// TIA Portal V15.1 export
// export: Created 2024-05-17T05:38:53.3669201Z, ExportSetting WithDefaults, DisplayName Totally Integrated Automation Portal, DisplayVersion V15.1 Update 5, DisplayName TIA Portal Openness, DisplayVersion V15.1 Update 5, DisplayName SINAMICS Startdrive Advanced, DisplayVersion V15.1, DisplayName G130, G150, S120, S150, SINAMICS MV, S210, DisplayVersion V15.1, DisplayName G110M, G120, G120C, G120D, G120P, DisplayVersion V15.1, DisplayName STEP 7 Professional, DisplayVersion V15.1 Update 5, DisplayName STEP 7 Safety, DisplayVersion V15.1, DisplayName WinCC Professional, DisplayVersion V15.1 Update 5, DisplayName SIMATIC Visualization Architect, DisplayVersion V15.1
FUNCTION_BLOCK "LGBCRComm"   // FB6692, FBD
TITLE = LGBCRComm
{ S7_Optimized_Access := 'TRUE' }
VERSION : 0.1
// stored: AutoNumber false, IsIECCheckEnabled false, IsRetainMemResEnabled false, MemoryReserve 100, SetENOAutomatically False, UDAEnableTagReadback false
   VAR_INPUT
      I_PlcActiveShift { ExternalAccessible := 'False'; ExternalVisible := 'False'; ExternalWritable := 'False'} : Int;
      I_PlcActiveBreak { ExternalAccessible := 'False'; ExternalVisible := 'False'; ExternalWritable := 'False'} : Int;
      I_StnAux01Feedback_Int { ExternalAccessible := 'False'; ExternalVisible := 'False'; ExternalWritable := 'False'} : Int;
      I_StnAux02Feedback_Int { ExternalAccessible := 'False'; ExternalVisible := 'False'; ExternalWritable := 'False'} : Int;
      I_StnAux03Feedback_Int { ExternalAccessible := 'False'; ExternalVisible := 'False'; ExternalWritable := 'False'} : Int;
      I_StnAux04Feedback_Int { ExternalAccessible := 'False'; ExternalVisible := 'False'; ExternalWritable := 'False'} : Int;
      I_StnAux05Feedback_Int { ExternalAccessible := 'False'; ExternalVisible := 'False'; ExternalWritable := 'False'} : Int;
      I_StnAux06Feedback_Int { ExternalAccessible := 'False'; ExternalVisible := 'False'; ExternalWritable := 'False'} : Int;
      I_StnAux07Feedback_DInt { ExternalAccessible := 'False'; ExternalVisible := 'False'; ExternalWritable := 'False'} : DInt;
      I_StnAux08Feedback_DInt { ExternalAccessible := 'False'; ExternalVisible := 'False'; ExternalWritable := 'False'} : DInt;
      I_StnAux09Feedback_DInt { ExternalAccessible := 'False'; ExternalVisible := 'False'; ExternalWritable := 'False'} : DInt;
      I_StnAux10Feedback_DInt { ExternalAccessible := 'False'; ExternalVisible := 'False'; ExternalWritable := 'False'} : DInt;
      I_StnAux11Feedback_DInt { ExternalAccessible := 'False'; ExternalVisible := 'False'; ExternalWritable := 'False'} : DInt;
      I_StnAux12Feedback_DInt { ExternalAccessible := 'False'; ExternalVisible := 'False'; ExternalWritable := 'False'} : DInt;
      I_StnAux13Feedback_Real { ExternalAccessible := 'False'; ExternalVisible := 'False'; ExternalWritable := 'False'} : Real;
      I_StnAux14Feedback_Real { ExternalAccessible := 'False'; ExternalVisible := 'False'; ExternalWritable := 'False'} : Real;
      I_StnAux15Feedback_Real { ExternalAccessible := 'False'; ExternalVisible := 'False'; ExternalWritable := 'False'} : Real;
      I_StnAux16Feedback_Real { ExternalAccessible := 'False'; ExternalVisible := 'False'; ExternalWritable := 'False'} : Real;
      I_StnAux17Feedback_Real { ExternalAccessible := 'False'; ExternalVisible := 'False'; ExternalWritable := 'False'} : Real;
      I_StnAux18Feedback_Real { ExternalAccessible := 'False'; ExternalVisible := 'False'; ExternalWritable := 'False'} : Real;
      C_DelayTimeAlarmC { ExternalAccessible := 'False'; ExternalVisible := 'False'; ExternalWritable := 'False'} : Time;
      C_DelayTimeAlarmD { ExternalAccessible := 'False'; ExternalVisible := 'False'; ExternalWritable := 'False'} : Time;
   END_VAR
   VAR_OUTPUT
      O_StnAux01_Int { ExternalAccessible := 'False'; ExternalVisible := 'False'; ExternalWritable := 'False'} : Int;
      O_StnAux02_Int { ExternalAccessible := 'False'; ExternalVisible := 'False'; ExternalWritable := 'False'} : Int;
      O_StnAux03_Int { ExternalAccessible := 'False'; ExternalVisible := 'False'; ExternalWritable := 'False'} : Int;
      O_StnAux04_Int { ExternalAccessible := 'False'; ExternalVisible := 'False'; ExternalWritable := 'False'} : Int;
      O_StnAux05_Int { ExternalAccessible := 'False'; ExternalVisible := 'False'; ExternalWritable := 'False'} : Int;
      O_StnAux06_Int { ExternalAccessible := 'False'; ExternalVisible := 'False'; ExternalWritable := 'False'} : Int;
      O_StnAux07_DInt { ExternalAccessible := 'False'; ExternalVisible := 'False'; ExternalWritable := 'False'} : DInt;
      O_StnAux08_DInt { ExternalAccessible := 'False'; ExternalVisible := 'False'; ExternalWritable := 'False'} : DInt;
      O_StnAux09_DInt { ExternalAccessible := 'False'; ExternalVisible := 'False'; ExternalWritable := 'False'} : DInt;
      O_StnAux10_DInt { ExternalAccessible := 'False'; ExternalVisible := 'False'; ExternalWritable := 'False'} : DInt;
      O_StnAux11_DInt { ExternalAccessible := 'False'; ExternalVisible := 'False'; ExternalWritable := 'False'} : DInt;
      O_StnAux12_DInt { ExternalAccessible := 'False'; ExternalVisible := 'False'; ExternalWritable := 'False'} : DInt;
      O_StnAux13_Real { ExternalAccessible := 'False'; ExternalVisible := 'False'; ExternalWritable := 'False'} : Real;
      O_StnAux14_Real { ExternalAccessible := 'False'; ExternalVisible := 'False'; ExternalWritable := 'False'} : Real;
      O_StnAux15_Real { ExternalAccessible := 'False'; ExternalVisible := 'False'; ExternalWritable := 'False'} : Real;
      O_StnAux16_Real { ExternalAccessible := 'False'; ExternalVisible := 'False'; ExternalWritable := 'False'} : Real;
      O_StnAux17_Real { ExternalAccessible := 'False'; ExternalVisible := 'False'; ExternalWritable := 'False'} : Real;
      O_StnAux18_Real { ExternalAccessible := 'False'; ExternalVisible := 'False'; ExternalWritable := 'False'} : Real;
   END_VAR
   VAR_IN_OUT
      IO_Modes : "Modes";   // Modes
      IO_DBZMToSv : "SupervisionZM";   // Send to supervision system
      IO_DBSvToZM : "SupervisionZM";   // Recieve from supervision system
   END_VAR
   VAR
      DelayAlarmC { ExternalAccessible := 'False'; ExternalVisible := 'False'; ExternalWritable := 'False'} : TON_TIME;
      DelayAlarmD { ExternalAccessible := 'False'; ExternalVisible := 'False'; ExternalWritable := 'False'} : TON_TIME;
      DelayUpperLevelZSAlarmC { ExternalAccessible := 'False'; ExternalVisible := 'False'; ExternalWritable := 'False'} : TON_TIME;
      DelayUpperLevelZSAlarmD { ExternalAccessible := 'False'; ExternalVisible := 'False'; ExternalWritable := 'False'} : TON_TIME;
      DelayUpperLevelPLCAlarmC { ExternalAccessible := 'False'; ExternalVisible := 'False'; ExternalWritable := 'False'} : TON_TIME;
      DelayUpperLevelPLCAlarmD { ExternalAccessible := 'False'; ExternalVisible := 'False'; ExternalWritable := 'False'} : TON_TIME;
   END_VAR
   VAR_TEMP
      Tmp_StnAux13Feedback_Real : Real;
      Tmp_StnAux14Feedback_Real : Real;
      Tmp_StnAux15Feedback_Real : Real;
      Tmp_StnAux16Feedback_Real : Real;
      Tmp_StnAux17Feedback_Real : Real;
      Tmp_StnAux18Feedback_Real : Real;
      Tmp_StnAux13_Real : Real;
      Tmp_StnAux14_Real : Real;
      Tmp_StnAux15_Real : Real;
      Tmp_StnAux16_Real : Real;
      Tmp_StnAux17_Real : Real;
      Tmp_StnAux18_Real : Real;
   END_VAR
BEGIN

REGION Network 1: **** 8 - Outputs **** Plc ActiveShift
   // Plc ActiveShift
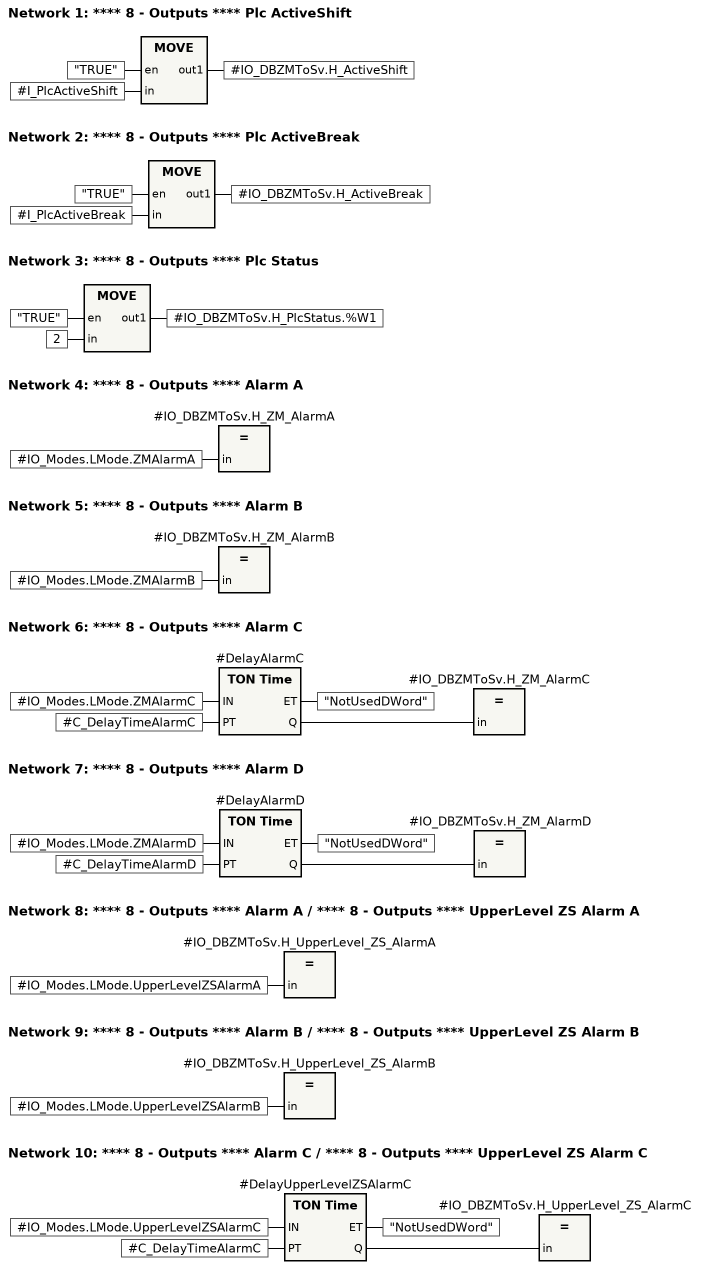
   IF "TRUE" THEN #IO_DBZMToSv.H_ActiveShift := #I_PlcActiveShift; END_IF;
END_REGION

REGION Network 2: **** 8 - Outputs **** Plc ActiveBreak
   // Plc ActiveBreak
   IF "TRUE" THEN #IO_DBZMToSv.H_ActiveBreak := #I_PlcActiveBreak; END_IF;
END_REGION

REGION Network 3: **** 8 - Outputs **** Plc Status
   // Plc Status
   IF "TRUE" THEN #IO_DBZMToSv.H_PlcStatus.%W1 := 2; END_IF;
END_REGION

REGION Network 4: **** 8 - Outputs **** Alarm A
   // Alarm A
   #IO_DBZMToSv.H_ZM_AlarmA := #IO_Modes.LMode.ZMAlarmA;
END_REGION

REGION Network 5: **** 8 - Outputs **** Alarm B
   // Alarm B
   #IO_DBZMToSv.H_ZM_AlarmB := #IO_Modes.LMode.ZMAlarmB;
END_REGION

REGION Network 6: **** 8 - Outputs **** Alarm C
   // Alarm C
   #DelayAlarmC(IN := #IO_Modes.LMode.ZMAlarmC, PT := #C_DelayTimeAlarmC, ET => "NotUsedDWord");   // TON
   #IO_DBZMToSv.H_ZM_AlarmC := #DelayAlarmC.Q;
END_REGION

REGION Network 7: **** 8 - Outputs **** Alarm D
   // Alarm D
   #DelayAlarmD(IN := #IO_Modes.LMode.ZMAlarmD, PT := #C_DelayTimeAlarmD, ET => "NotUsedDWord");   // TON
   #IO_DBZMToSv.H_ZM_AlarmD := #DelayAlarmD.Q;
END_REGION

REGION Network 8: **** 8 - Outputs **** Alarm A / **** 8 - Outputs **** UpperLevel ZS Alarm A
   // Alarm A
   #IO_DBZMToSv.H_UpperLevel_ZS_AlarmA := #IO_Modes.LMode.UpperLevelZSAlarmA;
END_REGION

REGION Network 9: **** 8 - Outputs **** Alarm B / **** 8 - Outputs **** UpperLevel ZS Alarm B
   // Alarm B
   #IO_DBZMToSv.H_UpperLevel_ZS_AlarmB := #IO_Modes.LMode.UpperLevelZSAlarmB;
END_REGION

REGION Network 10: **** 8 - Outputs **** Alarm C / **** 8 - Outputs **** UpperLevel ZS Alarm C
   // Alarm C
   #DelayUpperLevelZSAlarmC(IN := #IO_Modes.LMode.UpperLevelZSAlarmC,   // TON
                           PT := #C_DelayTimeAlarmC,
                           ET => "NotUsedDWord");
   #IO_DBZMToSv.H_UpperLevel_ZS_AlarmC := #DelayUpperLevelZSAlarmC.Q;
END_REGION

REGION Network 11: **** 8 - Outputs **** Alarm D / **** 8 - Outputs **** UpperLevel ZS Alarm D
   // Alarm D
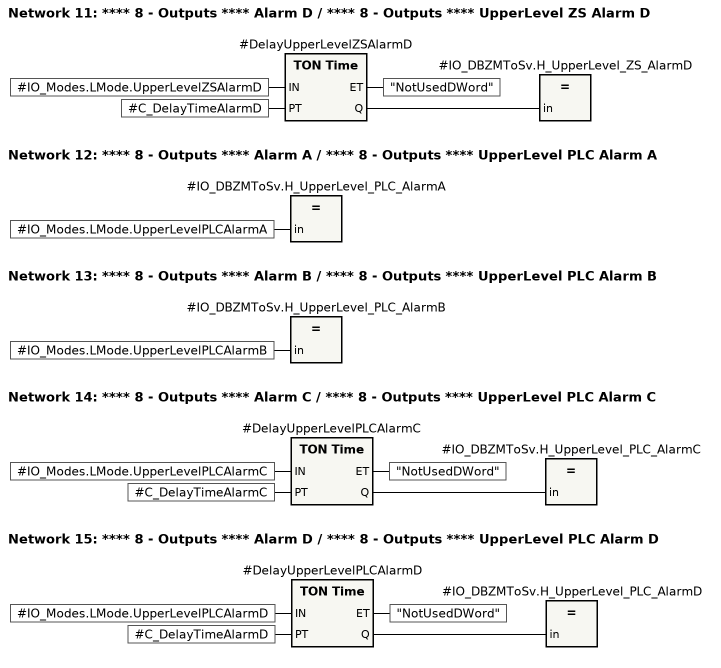
   #DelayUpperLevelZSAlarmD(IN := #IO_Modes.LMode.UpperLevelZSAlarmD,   // TON
                           PT := #C_DelayTimeAlarmD,
                           ET => "NotUsedDWord");
   #IO_DBZMToSv.H_UpperLevel_ZS_AlarmD := #DelayUpperLevelZSAlarmD.Q;
END_REGION

REGION Network 12: **** 8 - Outputs **** Alarm A / **** 8 - Outputs **** UpperLevel PLC Alarm A
   // Alarm A
   #IO_DBZMToSv.H_UpperLevel_PLC_AlarmA := #IO_Modes.LMode.UpperLevelPLCAlarmA;
END_REGION

REGION Network 13: **** 8 - Outputs **** Alarm B / **** 8 - Outputs **** UpperLevel PLC Alarm B
   // Alarm B
   #IO_DBZMToSv.H_UpperLevel_PLC_AlarmB := #IO_Modes.LMode.UpperLevelPLCAlarmB;
END_REGION

REGION Network 14: **** 8 - Outputs **** Alarm C / **** 8 - Outputs **** UpperLevel PLC Alarm C
   // Alarm C
   #DelayUpperLevelPLCAlarmC(IN := #IO_Modes.LMode.UpperLevelPLCAlarmC,   // TON
                           PT := #C_DelayTimeAlarmC,
                           ET => "NotUsedDWord");
   #IO_DBZMToSv.H_UpperLevel_PLC_AlarmC := #DelayUpperLevelPLCAlarmC.Q;
END_REGION

REGION Network 15: **** 8 - Outputs **** Alarm D / **** 8 - Outputs **** UpperLevel PLC Alarm D
   // Alarm D
   #DelayUpperLevelPLCAlarmD(IN := #IO_Modes.LMode.UpperLevelPLCAlarmD,   // TON
                           PT := #C_DelayTimeAlarmD,
                           ET => "NotUsedDWord");
   #IO_DBZMToSv.H_UpperLevel_PLC_AlarmD := #DelayUpperLevelPLCAlarmD.Q;
END_REGION

REGION Network 16: **** 8 - Outputs **** Operation Mode
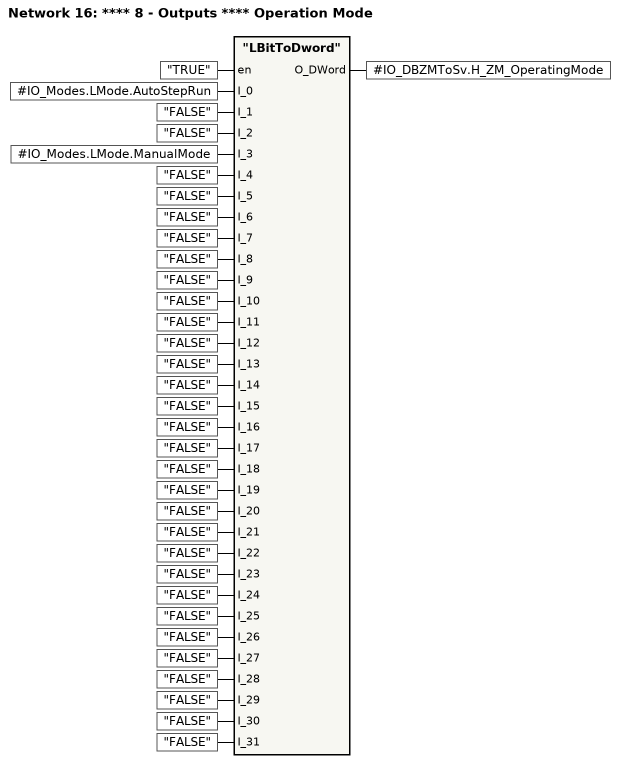
   IF "TRUE" THEN
       "LBitToDword"(I_0 := #IO_Modes.LMode.AutoStepRun,
                     I_1 := "FALSE",
                     I_2 := "FALSE",
                     I_3 := #IO_Modes.LMode.ManualMode,
                     I_4 := "FALSE",
                     I_5 := "FALSE",
                     I_6 := "FALSE",
                     I_7 := "FALSE",
                     I_8 := "FALSE",
                     I_9 := "FALSE",
                     I_10 := "FALSE",
                     I_11 := "FALSE",
                     I_12 := "FALSE",
                     I_13 := "FALSE",
                     I_14 := "FALSE",
                     I_15 := "FALSE",
                     I_16 := "FALSE",
                     I_17 := "FALSE",
                     I_18 := "FALSE",
                     I_19 := "FALSE",
                     I_20 := "FALSE",
                     I_21 := "FALSE",
                     I_22 := "FALSE",
                     I_23 := "FALSE",
                     I_24 := "FALSE",
                     I_25 := "FALSE",
                     I_26 := "FALSE",
                     I_27 := "FALSE",
                     I_28 := "FALSE",
                     I_29 := "FALSE",
                     I_30 := "FALSE",
                     I_31 := "FALSE",
                     O_DWord => #IO_DBZMToSv.H_ZM_OperatingMode);
   END_IF;
END_REGION

REGION Network 17: **** 8 - Outputs **** Operation Mode Sel
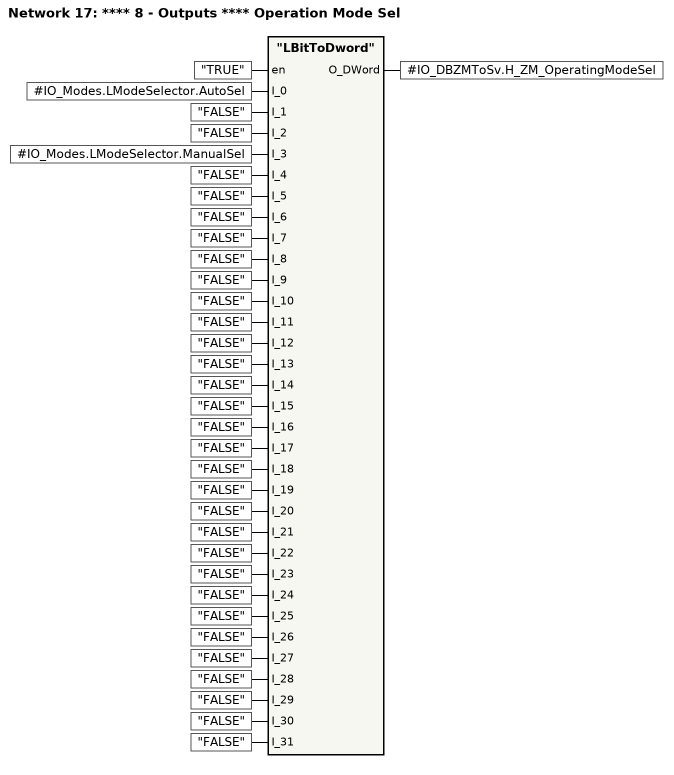
   IF "TRUE" THEN
       "LBitToDword"(I_0 := #IO_Modes.LModeSelector.AutoSel,
                     I_1 := "FALSE",
                     I_2 := "FALSE",
                     I_3 := #IO_Modes.LModeSelector.ManualSel,
                     I_4 := "FALSE",
                     I_5 := "FALSE",
                     I_6 := "FALSE",
                     I_7 := "FALSE",
                     I_8 := "FALSE",
                     I_9 := "FALSE",
                     I_10 := "FALSE",
                     I_11 := "FALSE",
                     I_12 := "FALSE",
                     I_13 := "FALSE",
                     I_14 := "FALSE",
                     I_15 := "FALSE",
                     I_16 := "FALSE",
                     I_17 := "FALSE",
                     I_18 := "FALSE",
                     I_19 := "FALSE",
                     I_20 := "FALSE",
                     I_21 := "FALSE",
                     I_22 := "FALSE",
                     I_23 := "FALSE",
                     I_24 := "FALSE",
                     I_25 := "FALSE",
                     I_26 := "FALSE",
                     I_27 := "FALSE",
                     I_28 := "FALSE",
                     I_29 := "FALSE",
                     I_30 := "FALSE",
                     I_31 := "FALSE",
                     O_DWord => #IO_DBZMToSv.H_ZM_OperatingModeSel);
   END_IF;
END_REGION

REGION Network 18: **** 8 - Outputs **** Production Mode
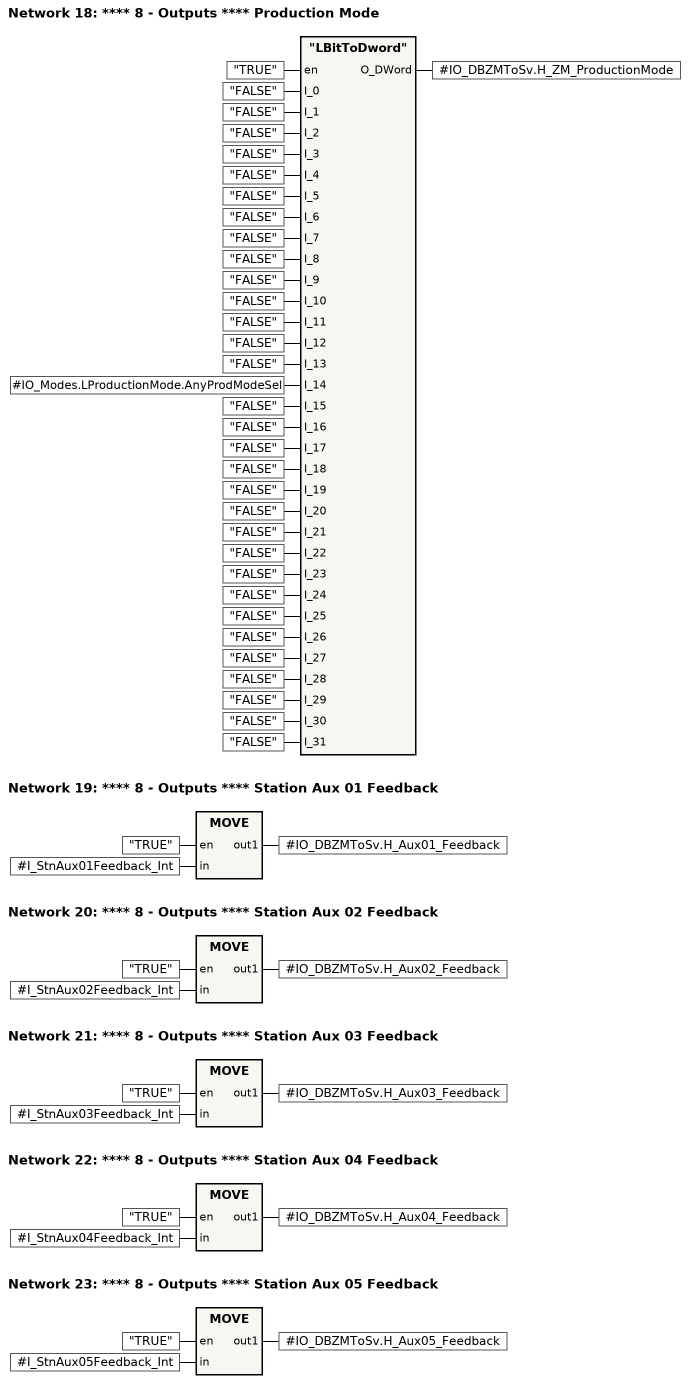
   IF "TRUE" THEN
       "LBitToDword"(I_0 := "FALSE",
                     I_1 := "FALSE",
                     I_2 := "FALSE",
                     I_3 := "FALSE",
                     I_4 := "FALSE",
                     I_5 := "FALSE",
                     I_6 := "FALSE",
                     I_7 := "FALSE",
                     I_8 := "FALSE",
                     I_9 := "FALSE",
                     I_10 := "FALSE",
                     I_11 := "FALSE",
                     I_12 := "FALSE",
                     I_13 := "FALSE",
                     I_14 := #IO_Modes.LProductionMode.AnyProdModeSel,
                     I_15 := "FALSE",
                     I_16 := "FALSE",
                     I_17 := "FALSE",
                     I_18 := "FALSE",
                     I_19 := "FALSE",
                     I_20 := "FALSE",
                     I_21 := "FALSE",
                     I_22 := "FALSE",
                     I_23 := "FALSE",
                     I_24 := "FALSE",
                     I_25 := "FALSE",
                     I_26 := "FALSE",
                     I_27 := "FALSE",
                     I_28 := "FALSE",
                     I_29 := "FALSE",
                     I_30 := "FALSE",
                     I_31 := "FALSE",
                     O_DWord => #IO_DBZMToSv.H_ZM_ProductionMode);
   END_IF;
END_REGION

REGION Network 19: **** 8 - Outputs **** Station Aux 01 Feedback
   // Station Aux 01 Feedback
   IF "TRUE" THEN #IO_DBZMToSv.H_Aux01_Feedback := #I_StnAux01Feedback_Int; END_IF;
END_REGION

REGION Network 20: **** 8 - Outputs **** Station Aux 02 Feedback
   // Station Aux 02 Feedback
   IF "TRUE" THEN #IO_DBZMToSv.H_Aux02_Feedback := #I_StnAux02Feedback_Int; END_IF;
END_REGION

REGION Network 21: **** 8 - Outputs **** Station Aux 03 Feedback
   // Station Aux 03 Feedback
   IF "TRUE" THEN #IO_DBZMToSv.H_Aux03_Feedback := #I_StnAux03Feedback_Int; END_IF;
END_REGION

REGION Network 22: **** 8 - Outputs **** Station Aux 04 Feedback
   // Station Aux 04 Feedback
   IF "TRUE" THEN #IO_DBZMToSv.H_Aux04_Feedback := #I_StnAux04Feedback_Int; END_IF;
END_REGION

REGION Network 23: **** 8 - Outputs **** Station Aux 05 Feedback
   // Station Aux 05 Feedback
   IF "TRUE" THEN #IO_DBZMToSv.H_Aux05_Feedback := #I_StnAux05Feedback_Int; END_IF;
END_REGION

REGION Network 24: **** 8 - Outputs **** Station Aux 06 Feedback
   // Station Aux 06 Feedback
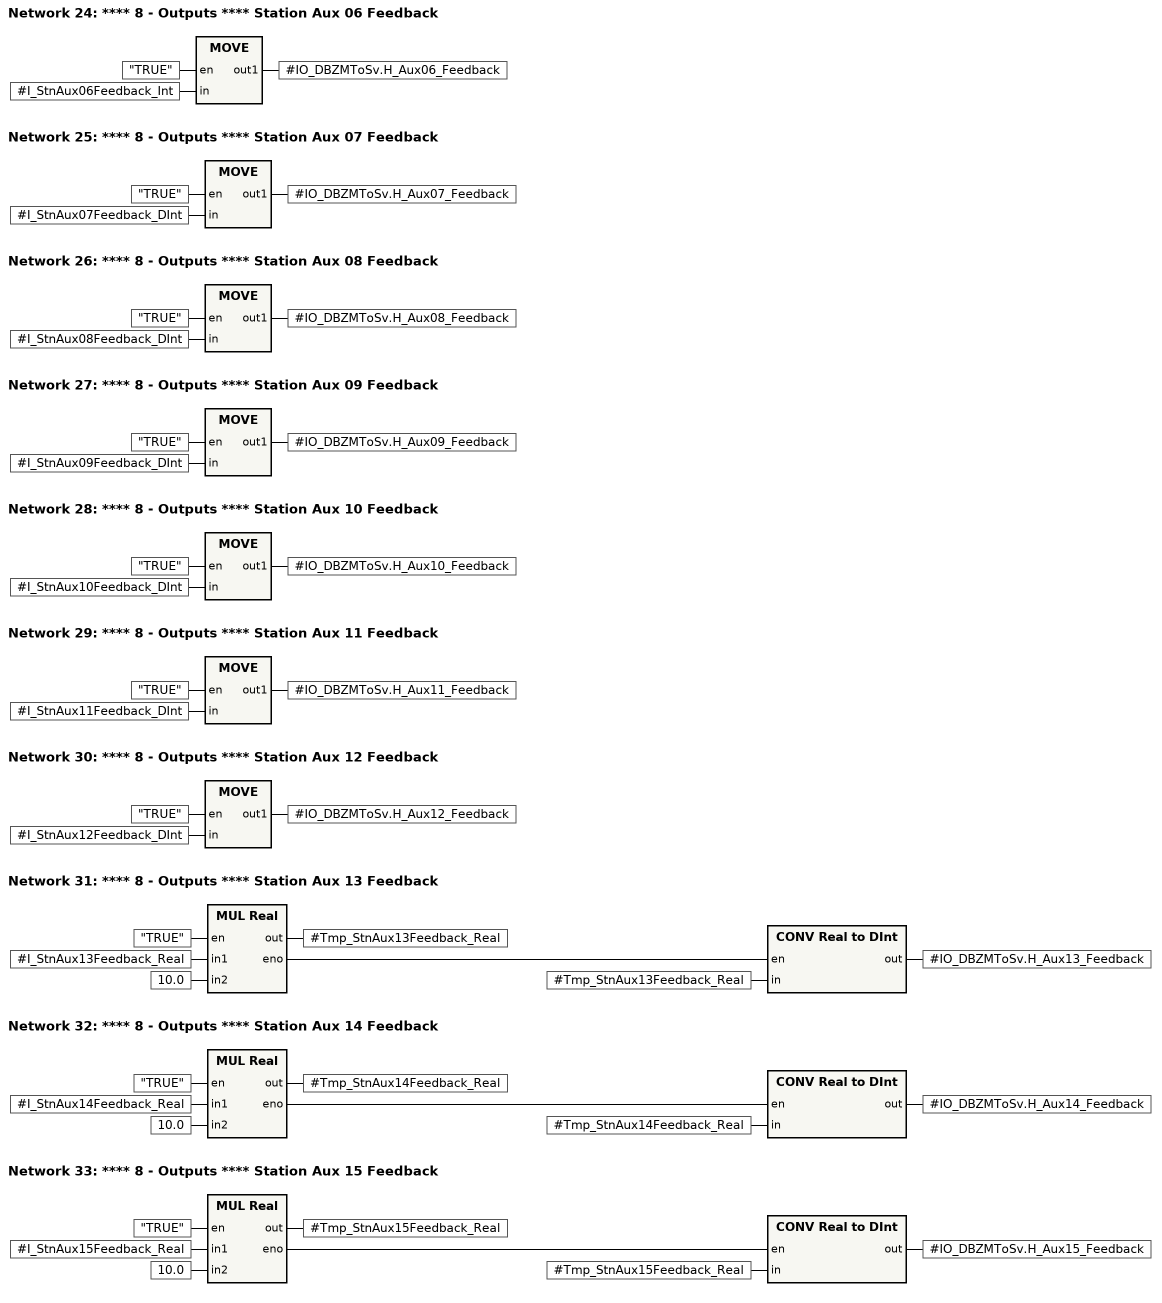
   IF "TRUE" THEN #IO_DBZMToSv.H_Aux06_Feedback := #I_StnAux06Feedback_Int; END_IF;
END_REGION

REGION Network 25: **** 8 - Outputs **** Station Aux 07 Feedback
   // Station Aux 07 Feedback
   IF "TRUE" THEN #IO_DBZMToSv.H_Aux07_Feedback := #I_StnAux07Feedback_DInt; END_IF;
END_REGION

REGION Network 26: **** 8 - Outputs **** Station Aux 08 Feedback
   // Station Aux 08 Feedback
   IF "TRUE" THEN #IO_DBZMToSv.H_Aux08_Feedback := #I_StnAux08Feedback_DInt; END_IF;
END_REGION

REGION Network 27: **** 8 - Outputs **** Station Aux 09 Feedback
   // Station Aux 09 Feedback
   IF "TRUE" THEN #IO_DBZMToSv.H_Aux09_Feedback := #I_StnAux09Feedback_DInt; END_IF;
END_REGION

REGION Network 28: **** 8 - Outputs **** Station Aux 10 Feedback
   // Station Aux 10 Feedback
   IF "TRUE" THEN #IO_DBZMToSv.H_Aux10_Feedback := #I_StnAux10Feedback_DInt; END_IF;
END_REGION

REGION Network 29: **** 8 - Outputs **** Station Aux 11 Feedback
   // Station Aux 11 Feedback
   IF "TRUE" THEN #IO_DBZMToSv.H_Aux11_Feedback := #I_StnAux11Feedback_DInt; END_IF;
END_REGION

REGION Network 30: **** 8 - Outputs **** Station Aux 12 Feedback
   // Station Aux 12 Feedback
   IF "TRUE" THEN #IO_DBZMToSv.H_Aux12_Feedback := #I_StnAux12Feedback_DInt; END_IF;
END_REGION

REGION Network 31: **** 8 - Outputs **** Station Aux 13 Feedback
   // Station Aux 13 Feedback
   IF "TRUE" THEN
       #Tmp_StnAux13Feedback_Real := #I_StnAux13Feedback_Real * 10.0;
       #IO_DBZMToSv.H_Aux13_Feedback := REAL_TO_DINT(#Tmp_StnAux13Feedback_Real);
   END_IF;
END_REGION

REGION Network 32: **** 8 - Outputs **** Station Aux 14 Feedback
   // Station Aux 14 Feedback
   IF "TRUE" THEN
       #Tmp_StnAux14Feedback_Real := #I_StnAux14Feedback_Real * 10.0;
       #IO_DBZMToSv.H_Aux14_Feedback := REAL_TO_DINT(#Tmp_StnAux14Feedback_Real);
   END_IF;
END_REGION

REGION Network 33: **** 8 - Outputs **** Station Aux 15 Feedback
   // Station Aux 15 Feedback
   IF "TRUE" THEN
       #Tmp_StnAux15Feedback_Real := #I_StnAux15Feedback_Real * 10.0;
       #IO_DBZMToSv.H_Aux15_Feedback := REAL_TO_DINT(#Tmp_StnAux15Feedback_Real);
   END_IF;
END_REGION

REGION Network 34: **** 8 - Outputs **** Station Aux 16 Feedback
   // Station Aux 16 Feedback
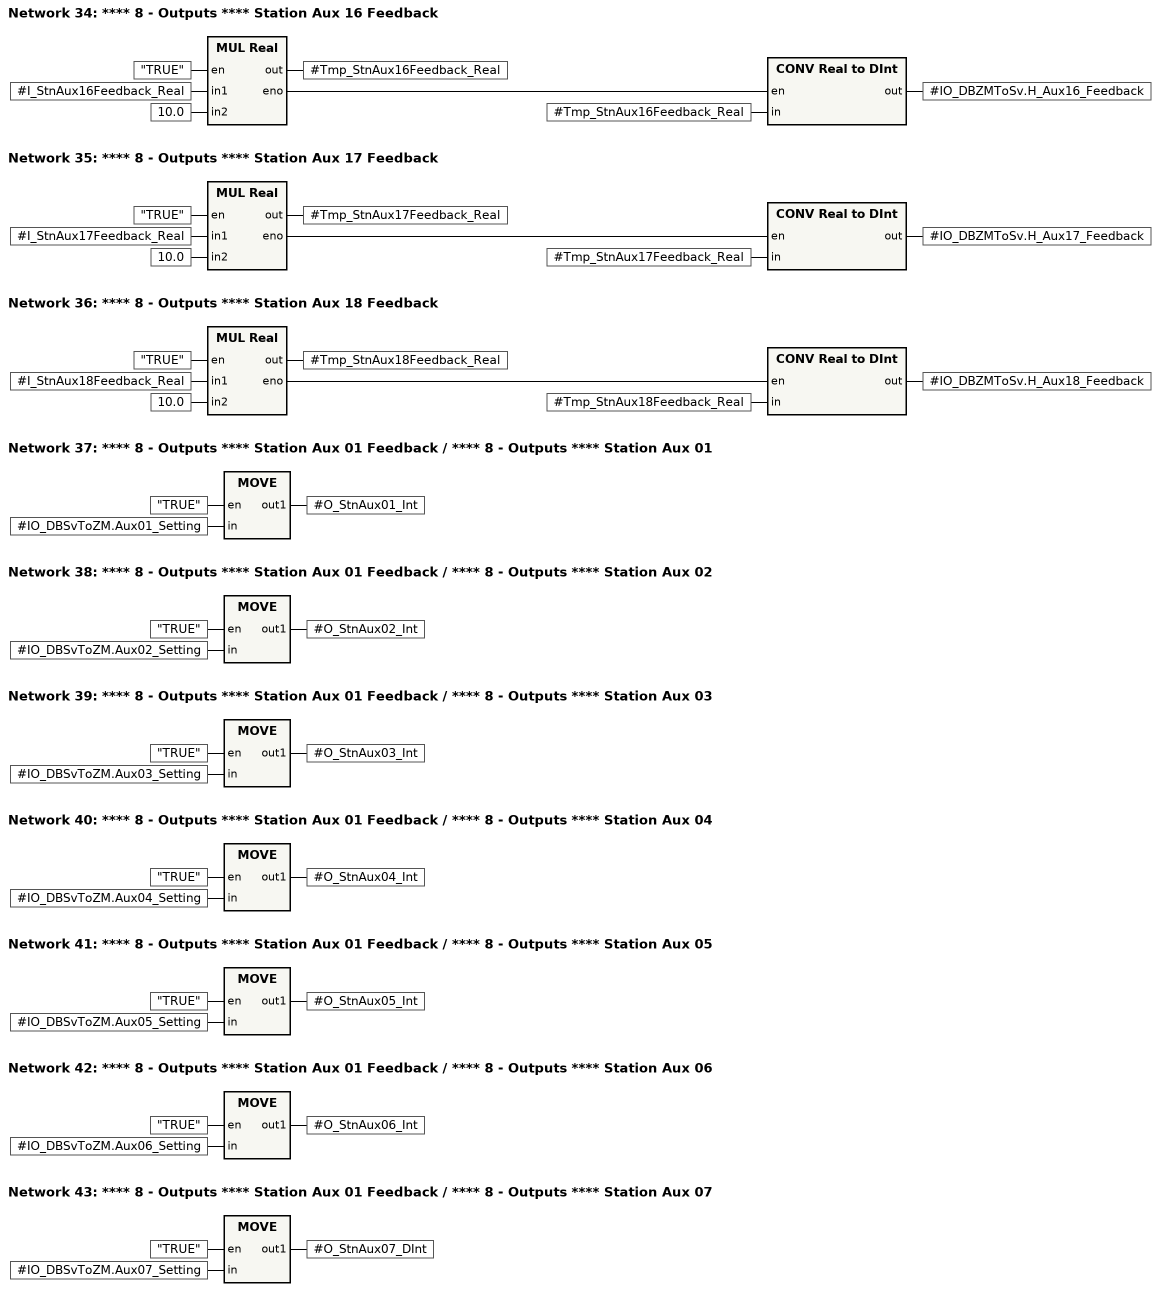
   IF "TRUE" THEN
       #Tmp_StnAux16Feedback_Real := #I_StnAux16Feedback_Real * 10.0;
       #IO_DBZMToSv.H_Aux16_Feedback := REAL_TO_DINT(#Tmp_StnAux16Feedback_Real);
   END_IF;
END_REGION

REGION Network 35: **** 8 - Outputs **** Station Aux 17 Feedback
   // Station Aux 17 Feedback
   IF "TRUE" THEN
       #Tmp_StnAux17Feedback_Real := #I_StnAux17Feedback_Real * 10.0;
       #IO_DBZMToSv.H_Aux17_Feedback := REAL_TO_DINT(#Tmp_StnAux17Feedback_Real);
   END_IF;
END_REGION

REGION Network 36: **** 8 - Outputs **** Station Aux 18 Feedback
   // Station Aux 18 Feedback
   IF "TRUE" THEN
       #Tmp_StnAux18Feedback_Real := #I_StnAux18Feedback_Real * 10.0;
       #IO_DBZMToSv.H_Aux18_Feedback := REAL_TO_DINT(#Tmp_StnAux18Feedback_Real);
   END_IF;
END_REGION

REGION Network 37: **** 8 - Outputs **** Station Aux 01 Feedback / **** 8 - Outputs **** Station Aux 01
   // Station Aux 01 Feedback / Station Aux 01
   IF "TRUE" THEN #O_StnAux01_Int := #IO_DBSvToZM.Aux01_Setting; END_IF;
END_REGION

REGION Network 38: **** 8 - Outputs **** Station Aux 01 Feedback / **** 8 - Outputs **** Station Aux 02
   // Station Aux 01 Feedback / Station Aux 02
   IF "TRUE" THEN #O_StnAux02_Int := #IO_DBSvToZM.Aux02_Setting; END_IF;
END_REGION

REGION Network 39: **** 8 - Outputs **** Station Aux 01 Feedback / **** 8 - Outputs **** Station Aux 03
   // Station Aux 01 Feedback / Station Aux 03
   IF "TRUE" THEN #O_StnAux03_Int := #IO_DBSvToZM.Aux03_Setting; END_IF;
END_REGION

REGION Network 40: **** 8 - Outputs **** Station Aux 01 Feedback / **** 8 - Outputs **** Station Aux 04
   // Station Aux 01 Feedback / Station Aux 04
   IF "TRUE" THEN #O_StnAux04_Int := #IO_DBSvToZM.Aux04_Setting; END_IF;
END_REGION

REGION Network 41: **** 8 - Outputs **** Station Aux 01 Feedback / **** 8 - Outputs **** Station Aux 05
   // Station Aux 01 Feedback / Station Aux 05
   IF "TRUE" THEN #O_StnAux05_Int := #IO_DBSvToZM.Aux05_Setting; END_IF;
END_REGION

REGION Network 42: **** 8 - Outputs **** Station Aux 01 Feedback / **** 8 - Outputs **** Station Aux 06
   // Station Aux 01 Feedback / Station Aux 06
   IF "TRUE" THEN #O_StnAux06_Int := #IO_DBSvToZM.Aux06_Setting; END_IF;
END_REGION

REGION Network 43: **** 8 - Outputs **** Station Aux 01 Feedback / **** 8 - Outputs **** Station Aux 07
   // Station Aux 01 Feedback / Station Aux 07
   IF "TRUE" THEN #O_StnAux07_DInt := #IO_DBSvToZM.Aux07_Setting; END_IF;
END_REGION

REGION Network 44: **** 8 - Outputs **** Station Aux 01 Feedback / **** 8 - Outputs **** Station Aux 08
   // Station Aux 01 Feedback / Station Aux 08
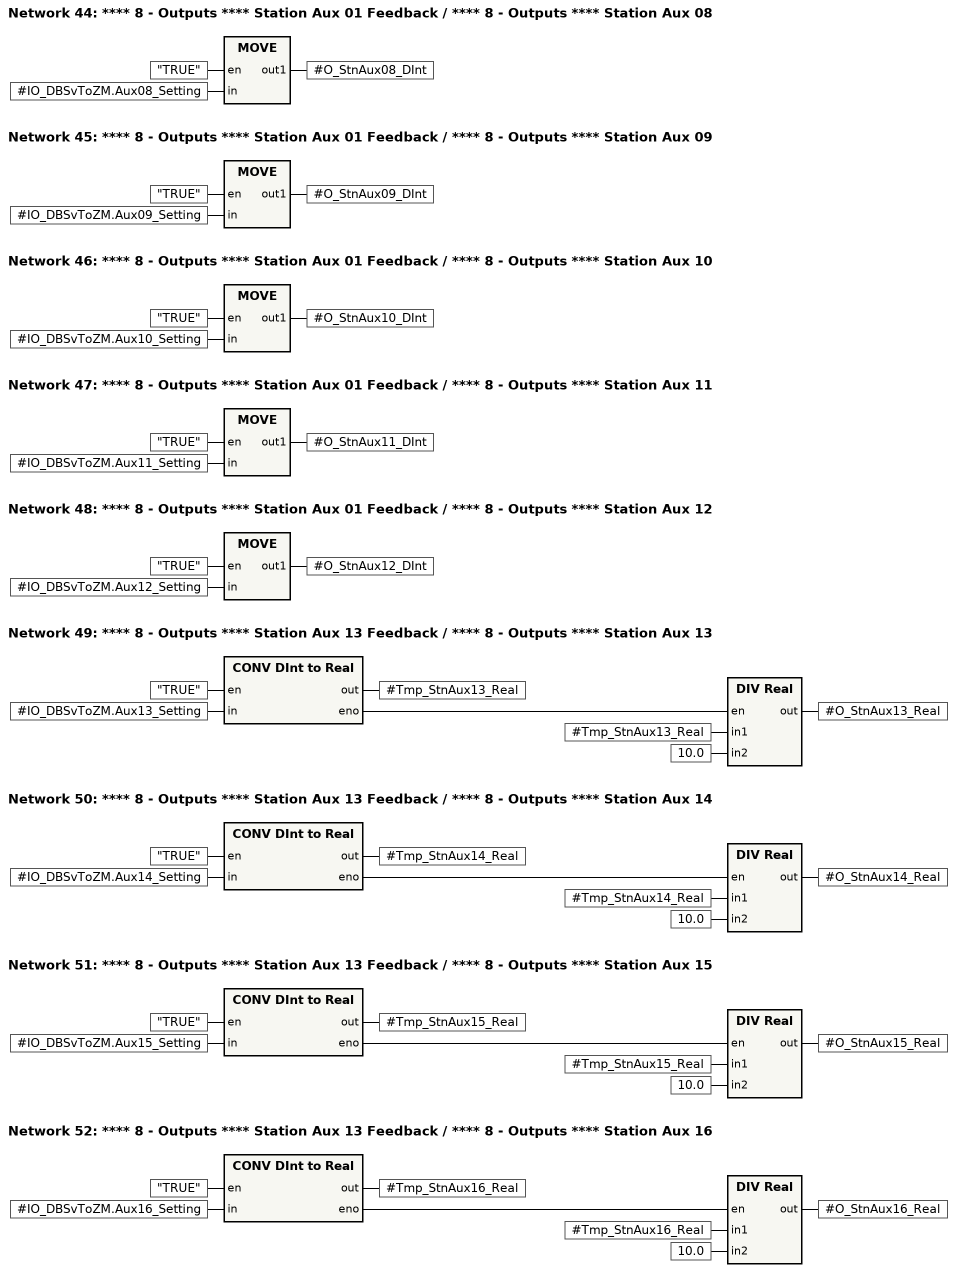
   IF "TRUE" THEN #O_StnAux08_DInt := #IO_DBSvToZM.Aux08_Setting; END_IF;
END_REGION

REGION Network 45: **** 8 - Outputs **** Station Aux 01 Feedback / **** 8 - Outputs **** Station Aux 09
   // Station Aux 01 Feedback / Station Aux 09
   IF "TRUE" THEN #O_StnAux09_DInt := #IO_DBSvToZM.Aux09_Setting; END_IF;
END_REGION

REGION Network 46: **** 8 - Outputs **** Station Aux 01 Feedback / **** 8 - Outputs **** Station Aux 10
   // Station Aux 01 Feedback / Station Aux 10
   IF "TRUE" THEN #O_StnAux10_DInt := #IO_DBSvToZM.Aux10_Setting; END_IF;
END_REGION

REGION Network 47: **** 8 - Outputs **** Station Aux 01 Feedback / **** 8 - Outputs **** Station Aux 11
   // Station Aux 01 Feedback / Station Aux 11
   IF "TRUE" THEN #O_StnAux11_DInt := #IO_DBSvToZM.Aux11_Setting; END_IF;
END_REGION

REGION Network 48: **** 8 - Outputs **** Station Aux 01 Feedback / **** 8 - Outputs **** Station Aux 12
   // Station Aux 01 Feedback / Station Aux 12
   IF "TRUE" THEN #O_StnAux12_DInt := #IO_DBSvToZM.Aux12_Setting; END_IF;
END_REGION

REGION Network 49: **** 8 - Outputs **** Station Aux 13 Feedback / **** 8 - Outputs **** Station Aux 13
   // Station Aux 13 Feedback / Station Aux 13
   IF "TRUE" THEN
       #Tmp_StnAux13_Real := DINT_TO_REAL(#IO_DBSvToZM.Aux13_Setting);
       #O_StnAux13_Real := #Tmp_StnAux13_Real / 10.0;
   END_IF;
END_REGION

REGION Network 50: **** 8 - Outputs **** Station Aux 13 Feedback / **** 8 - Outputs **** Station Aux 14
   // Station Aux 13 Feedback / Station Aux 14
   IF "TRUE" THEN
       #Tmp_StnAux14_Real := DINT_TO_REAL(#IO_DBSvToZM.Aux14_Setting);
       #O_StnAux14_Real := #Tmp_StnAux14_Real / 10.0;
   END_IF;
END_REGION

REGION Network 51: **** 8 - Outputs **** Station Aux 13 Feedback / **** 8 - Outputs **** Station Aux 15
   // Station Aux 13 Feedback / Station Aux 15
   IF "TRUE" THEN
       #Tmp_StnAux15_Real := DINT_TO_REAL(#IO_DBSvToZM.Aux15_Setting);
       #O_StnAux15_Real := #Tmp_StnAux15_Real / 10.0;
   END_IF;
END_REGION

REGION Network 52: **** 8 - Outputs **** Station Aux 13 Feedback / **** 8 - Outputs **** Station Aux 16
   // Station Aux 13 Feedback / Station Aux 16
   IF "TRUE" THEN
       #Tmp_StnAux16_Real := DINT_TO_REAL(#IO_DBSvToZM.Aux16_Setting);
       #O_StnAux16_Real := #Tmp_StnAux16_Real / 10.0;
   END_IF;
END_REGION

REGION Network 53: **** 8 - Outputs **** Station Aux 13 Feedback / **** 8 - Outputs **** Station Aux 17
   // Station Aux 13 Feedback / Station Aux 17
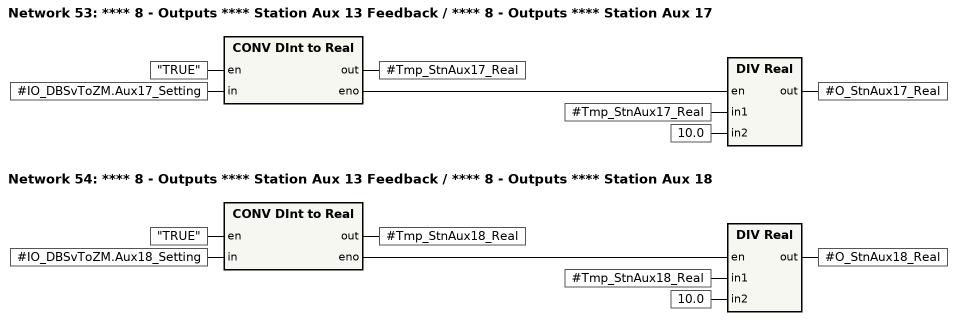
   IF "TRUE" THEN
       #Tmp_StnAux17_Real := DINT_TO_REAL(#IO_DBSvToZM.Aux17_Setting);
       #O_StnAux17_Real := #Tmp_StnAux17_Real / 10.0;
   END_IF;
END_REGION

REGION Network 54: **** 8 - Outputs **** Station Aux 13 Feedback / **** 8 - Outputs **** Station Aux 18
   // Station Aux 13 Feedback / Station Aux 18
   IF "TRUE" THEN
       #Tmp_StnAux18_Real := DINT_TO_REAL(#IO_DBSvToZM.Aux18_Setting);
       #O_StnAux18_Real := #Tmp_StnAux18_Real / 10.0;
   END_IF;
END_REGION
END_FUNCTION_BLOCK
